Staubli VAL3: goToPoint.pgx

program goToPoint()
begin
  logMsg("  goToPoint start")

  if(bPinceOpen == true)
    open(tTool)
  else
    close(tTool)
  endIf


  movel(pTarget, tTool, mRapide100)

  waitEndMove()

  bAcquisitionOk = false
end
